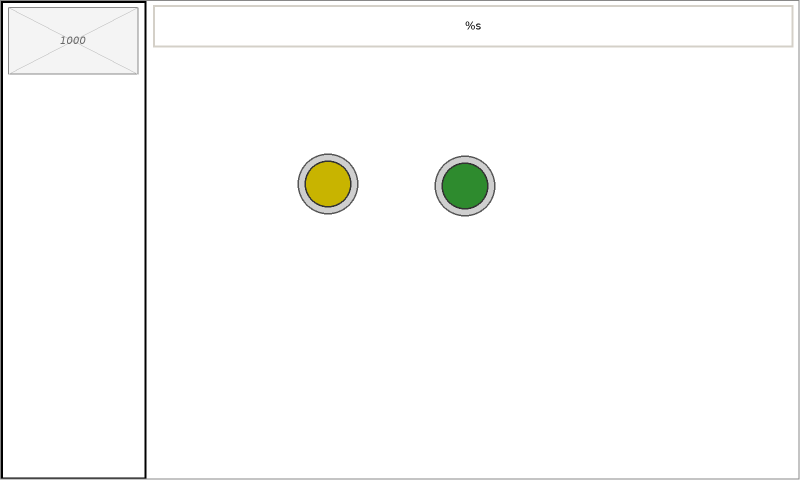
VISUALIZATION Visualization  // 800x480
    Rectangle (1,1 145x478)
    Lamp1 (430,151 70x70), variable: GVL.SET_TEST_OUTPUT, style: Lamp-Lamp1-Green
    Lamp1 (293,149 70x70), variable: GVL.SET_TEST_OUTPUT, style: Lamp-Lamp1-Yellow
    Textfield (153,5 640x42), "%s", text variable: GVL.RFID_TAG
    Image (8,7 130x67), image: 1000
END_VISUALIZATION

(* stored: Version 1.1.0.1, ProductVersion 3.1.4020.6
   Visu Visualization: Id {74244b8a-fd06-4c16-88e6-d991d6c70988} *)
